{attribute addProperty BoxType "AMP8000-0030-0103-0103"}
{attribute addProperty Id "WcState0AT %I*BOOL810WcState1AT %I*BOOL810InputToggle0AT %I*BOOL810InputToggle1AT %I*BOOL810"}
{attribute addProperty CRC "3249998607"}
{attribute addProperty SizeInBites "32"}
{attribute addProperty SizeInBytes "4"}
TYPE WcState_C1B70B0F :
STRUCT
	{attribute addProperty Name "WcState0"}
	WcState0 AT %I* : BOOL;
	{attribute addProperty Name "WcState1"}
	WcState1 AT %I* : BOOL;
	{attribute addProperty Name "InputToggle0"}
	InputToggle0 AT %I* : BOOL;
	{attribute addProperty Name "InputToggle1"}
	InputToggle1 AT %I* : BOOL;
END_STRUCT
END_TYPE

(* stored: Version 1.2.0.0, ProductVersion 3.1.4024.9
   DUT WcState_C1B70B0F: Id {d2a03e8d-dab1-4805-8461-94005d472094} *)
